Universal Robots PolyScope program: flip_endcap.urp

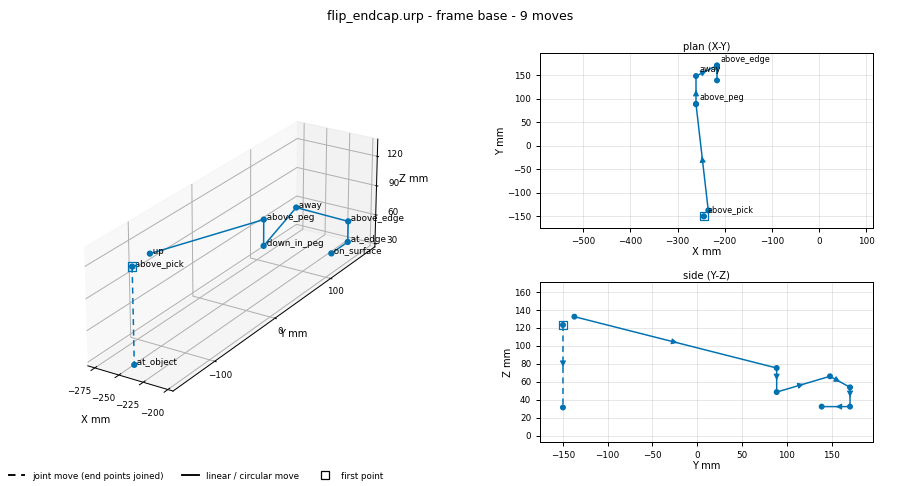
[picture p0: tool path of flip_endcap.urp in frame base, 9 of 14 moves have a stored position in this frame; points joined in program order, loops and branches not executed]
Program flip_endcap (installation=default directory=/programs/wrs2020 createdIn=5.7.0.90932 lastSavedIn=5.9.1.1031110 robotSerialNumber=20205500180)
Calibrated DH parameters: a=[0, -0.425, -0.3922, 0, 0, 0]; d=[0.1625, 0, 0, 0.1333, 0.0997, 0.0996]; alpha=[1.570796, 0, 0, 1.570796, -1.570796, 0]; deltaTheta=[0, 0, 0, 0, 0, 0]
Robot Program (runOnlyOnce=true)
  MoveJ speed 60 deg/s, acceleration 80 deg/s^2 (useActiveTCP=true) feature=Base
    currentpose := get_actual_tcp_pose()get_actual_joint_positions()
    Waypoint Waypoint (Variable): variable=currentpose
  URCap Gripper (Robotiq_Grippers, Robotiq Inc.) dataModel(position=56.470588235294116, force=100.0, speed=0.0, positionInDouble=56.470588235294116, forceInDouble=100.0, speedInDouble=0.0, slaveIds=[9], blocking=true)
  MoveJ speed 60 deg/s, acceleration 80 deg/s^2 (useActiveTCP=true) feature=Base
    Waypoint above_pick: TCP in base x=-244.307 y=-149.766 z=123.376 mm, rx=2.1485 ry=2.2672 rz=0.0007 rad; joints [2.86, -122.568, 133.81, -100.505, -89.267, -0.224] deg; TCP offset x=0 y=0 z=220 mm, rx=0 ry=0 rz=0 rad
    Waypoint at_object: TCP in base x=-244.319 y=-149.767 z=31.341 mm, rx=2.1485 ry=2.2672 rz=0.0007 rad; joints [2.86, -115.916, 145.325, -118.672, -89.267, -0.225] deg
  Folder center_object
    URCap Gripper (Robotiq_Grippers, Robotiq Inc.) dataModel(position=100.0, force=0.0, speed=0.0, positionInDouble=100.0, forceInDouble=0.0, speedInDouble=0.0, slaveIds=[9], blocking=true)
    URCap Gripper (Robotiq_Grippers, Robotiq Inc.) dataModel(position=56.470588235294116, force=100.0, speed=0.0, positionInDouble=56.470588235294116, forceInDouble=100.0, speedInDouble=0.0, slaveIds=[9], blocking=true)
    MoveJ speed 180 deg/s, acceleration 800 deg/s^2 (useActiveTCP=true) feature=Base
      Waypoint turn_right (Relative): relativeFromPosition TCP in base x=218.277 y=-500.897 z=48.153 mm, rx=-2.1842 ry=2.228 rz=-0.024 rad; joints [98.784, -72.216, 112.616, -130.369, -88.16, -80.001] deg; TCP offset x=0 y=0 z=165 mm, rx=0 ry=0 rz=0 rad; TCP in base x=218.316 y=-500.86 z=48.143 mm, rx=0.031 ry=3.1153 rz=0.0068 rad; joints [98.786, -72.217, 112.618, -130.367, -88.154, 10.001] deg
    URCap Gripper (Robotiq_Grippers, Robotiq Inc.) dataModel(position=100.0, force=0.0, speed=0.0, positionInDouble=100.0, forceInDouble=0.0, speedInDouble=0.0, slaveIds=[9], blocking=true)
    URCap Gripper (Robotiq_Grippers, Robotiq Inc.) dataModel(position=56.470588235294116, force=100.0, speed=0.0, positionInDouble=56.470588235294116, forceInDouble=100.0, speedInDouble=0.0, slaveIds=[9], blocking=true)
    MoveJ speed 180 deg/s, acceleration 1000 deg/s^2 (useActiveTCP=true) feature=Base
      Waypoint turn_left (Relative): relativeFromPosition TCP in base x=218.287 y=-500.864 z=48.112 mm, rx=0.031 ry=3.1154 rz=0.0069 rad; joints [98.785, -72.214, 112.618, -130.367, -88.158, 9.999] deg; TCP in base x=218.294 y=-500.846 z=48.105 mm, rx=-2.1841 ry=2.228 rz=-0.0238 rad; joints [98.786, -72.214, 112.619, -130.366, -88.158, -79.999] deg
    URCap Gripper (Robotiq_Grippers, Robotiq Inc.) dataModel(position=100.0, force=0.0, speed=0.0, positionInDouble=100.0, forceInDouble=0.0, speedInDouble=0.0, slaveIds=[9], blocking=true)
  MoveL speed 50 mm/s, acceleration 1200 mm/s^2 (useActiveTCP=true) feature=Base
    Waypoint up: TCP in base x=-234.858 y=-137.043 z=132.633 mm, rx=2.0849 ry=2.3425 rz=-0.0345 rad; joints [-0.668, -127.537, 134.623, -97.675, -88.84, -7.322] deg; TCP offset x=0 y=0 z=220 mm, rx=0 ry=0 rz=0 rad
    Waypoint above_peg: motionParameters(jointSpeed=1.047198 jointAcceleration=1.396263 cartesianSpeed=0.25 cartesianAcceleration=1.2); TCP in base x=-260.868 y=88.598 z=75.369 mm, rx=-3.1387 ry=-0.0312 rz=0.0402 rad; joints [-49.061, -124.602, 142.312, -108.77, -88.976, 39.809] deg
    Waypoint down_in_peg: motionParameters(jointSpeed=1.047198 jointAcceleration=1.396263 cartesianSpeed=0.005 cartesianAcceleration=0.01); TCP in base x=-260.887 y=88.608 z=48.514 mm, rx=-3.1386 ry=-0.0312 rz=0.0402 rad; joints [-49.061, -122.443, 145.723, -114.343, -88.975, 39.81] deg
    Waypoint away: motionParameters(jointSpeed=1.047198 jointAcceleration=1.396263 cartesianSpeed=0.25 cartesianAcceleration=1.2); TCP in base x=-260.867 y=148.093 z=66.133 mm, rx=-3.1387 ry=-0.0312 rz=0.0402 rad; joints [-57.363, -118.12, 141.124, -113.903, -88.833, -328.494] deg
    Waypoint above_edge: motionParameters(jointSpeed=1.047198 jointAcceleration=1.396263 cartesianSpeed=0.8 cartesianAcceleration=0.8); TCP in base x=-216.31 y=170.428 z=53.803 mm, rx=0.1308 ry=3.1245 rz=-0.0139 rad; joints [-66.502, -120.005, 143.405, -112.583, -90.517, -151.705] deg
    Waypoint at_edge: TCP in base x=-216.291 y=170.399 z=32.316 mm, rx=0.1307 ry=3.1244 rz=-0.0141 rad; joints [-66.5, -117.824, 145.978, -117.329, -90.519, -151.705] deg
    Waypoint on_surface: motionParameters(jointSpeed=1.047198 jointAcceleration=1.396263 cartesianSpeed=0.01 cartesianAcceleration=0.01); TCP in base x=-216.285 y=138.807 z=32.315 mm, rx=0.1308 ry=3.1244 rz=-0.0141 rad; joints [-63.252, -122.469, 147.785, -114.461, -90.472, -148.455] deg
  URCap Gripper (Robotiq_Grippers, Robotiq Inc.) dataModel(position=56.470588235294116, force=100.0, speed=0.0, positionInDouble=56.470588235294116, forceInDouble=100.0, speedInDouble=0.0, slaveIds=[9], blocking=true)
  Folder center_object
    URCap Gripper (Robotiq_Grippers, Robotiq Inc.) dataModel(position=100.0, force=0.0, speed=0.0, positionInDouble=100.0, forceInDouble=0.0, speedInDouble=0.0, slaveIds=[9], blocking=true)
    URCap Gripper (Robotiq_Grippers, Robotiq Inc.) dataModel(position=56.470588235294116, force=100.0, speed=0.0, positionInDouble=56.470588235294116, forceInDouble=100.0, speedInDouble=0.0, slaveIds=[9], blocking=true)
    MoveJ speed 180 deg/s, acceleration 800 deg/s^2 (useActiveTCP=true) feature=Base
      Waypoint turn_right (Relative): relativeFromPosition TCP in base x=218.277 y=-500.897 z=48.153 mm, rx=-2.1842 ry=2.228 rz=-0.024 rad; joints [98.784, -72.216, 112.616, -130.369, -88.16, -80.001] deg; TCP offset x=0 y=0 z=165 mm, rx=0 ry=0 rz=0 rad; TCP in base x=218.316 y=-500.86 z=48.143 mm, rx=0.031 ry=3.1153 rz=0.0068 rad; joints [98.786, -72.217, 112.618, -130.367, -88.154, 10.001] deg
    URCap Gripper (Robotiq_Grippers, Robotiq Inc.) dataModel(position=100.0, force=0.0, speed=0.0, positionInDouble=100.0, forceInDouble=0.0, speedInDouble=0.0, slaveIds=[9], blocking=true)
    URCap Gripper (Robotiq_Grippers, Robotiq Inc.) dataModel(position=56.470588235294116, force=100.0, speed=0.0, positionInDouble=56.470588235294116, forceInDouble=100.0, speedInDouble=0.0, slaveIds=[9], blocking=true)
    MoveJ speed 180 deg/s, acceleration 1000 deg/s^2 (useActiveTCP=true) feature=Base
      Waypoint turn_left (Relative): relativeFromPosition TCP in base x=218.287 y=-500.864 z=48.112 mm, rx=0.031 ry=3.1154 rz=0.0069 rad; joints [98.785, -72.214, 112.618, -130.367, -88.158, 9.999] deg; TCP in base x=218.294 y=-500.846 z=48.105 mm, rx=-2.1841 ry=2.228 rz=-0.0238 rad; joints [98.786, -72.214, 112.619, -130.366, -88.158, -79.999] deg
    URCap Gripper (Robotiq_Grippers, Robotiq Inc.) dataModel(position=100.0, force=0.0, speed=0.0, positionInDouble=100.0, forceInDouble=0.0, speedInDouble=0.0, slaveIds=[9], blocking=true)
  MoveL speed 50 mm/s, acceleration 1200 mm/s^2 (useActiveTCP=true) feature=Base
    MoveDirectionNode (selectedDirection=ZPlus)
      Until DISTANCE (allowActions=false deceleration=3 distanceNodeType=STOP) Distance=0.05; motionParameters(blendRadius=0)
